PROGRAM P_Demo_FB_MBWriteCoils
VAR
    fbWriteCoils  : FB_MBWriteCoils;
    sTargetIp     : STRING(15) := '192.168.1.50';   // 目标 Modbus 设备 IP（按现场改）
    bTrigger      : BOOL;          // 在线置一次上升沿触发本次访问
    bBusy         : BOOL;          // 在线 monitor：执行中为 TRUE
    bError        : BOOL;          // 出错置 TRUE
    nErrId        : UDINT;         // 出错时的 ADS/Modbus 错误码
    arrData       : ARRAY [0..1] OF BYTE := [16#75,16#03];   // 待写出的数据
END_VAR

// ============================================================
// Tc2_ModbusSrv.FB_MBWriteCoils 演示程序（Modbus TCP 客户端 / 主站）
// ============================================================
// 场景：一次性下发一批继电器/输出状态，例如远端 IO 站的 10 路输出按一个 `BYTE` 模式批量置位，用于灯光/电磁阀阵列控制。
// 价值：批量写线圈用功能码 15，比逐个功能码 5 少很多报文往返；本 FB 按位打包一次写出。
// 验证：登录后在线置 bTrigger := TRUE 触发一次；观察 bBusy 在数个周期后回 FALSE，
//       bError 应为 FALSE、nErrId 应为 0；若对端不在线则 bError=TRUE 且 nErrId 含超时码。
//       本例：一次写 10 个线圈，位模式 0x0375 的低 10 位
// 验证步骤：
//   1. 右键 PLC 项目下 POUs 文件夹 → Add → Existing Item → 选本 .TcPOU 文件
//   2. 引用 Tc2_ModbusSrv（References → Add library），并确保 TF6250 Modbus TCP 已授权运行
//   3. 把 sTargetIp 改成现场 Modbus 设备 IP；编译 → 登录 → 运行
//   4. 在线脉冲 bTrigger，按上方『验证』观察输出
// ============================================================

// 单次完整调用：所有 VAR_INPUT 显式赋值；bExecute 边沿触发一次
fbWriteCoils(
    sIPAddr   := sTargetIp,
    nTCPPort  := MODBUS_TCP_PORT,
    nUnitID   := 16#FF,
    nQuantity := 10,
    nMBAddr   := 0,
    cbLength  := SIZEOF(arrData),
    pSrcAddr  := ADR(arrData),
    bExecute  := bTrigger,
    tTimeout  := T#5S,
    bBUSY     => bBusy,
    bError    => bError,
    nErrId    => nErrId
);

END_PROGRAM

(* stored: Version 1.1.0.1, ProductVersion 3.1.4024.5
   POU P_Demo_FB_MBWriteCoils: Id {384fa515-1e74-531a-b12a-12ebe203bf18}, SpecialFunc None *)
